// TwinCAT 3 PLC project Untitled1
// ProgramVersion: 3.1.4022.3
// libraries:
//   Tc2_Standard, * (Beckhoff Automation GmbH)
//   Tc2_System, * (Beckhoff Automation GmbH)
//   Tc3_Module, * (Beckhoff Automation GmbH)
// project tree:
//   / PlcTask.TcTTO
//   POUs/ FC1.TcPOU, FC2.TcPOU, FC3.TcPOU, MAIN.TcPOU

CONFIGURATION Untitled1
    RESOURCE PLC ON TwinCAT3
        TASK PlcTask(INTERVAL := T#10ms, PRIORITY := 20);
        PROGRAM MAIN WITH PlcTask : MAIN;
    END_RESOURCE
END_CONFIGURATION

// ---- POUs/MAIN.TcPOU
PROGRAM MAIN
VAR
  test :INT;
  test1 :INT;
  test2 :INT;
  test3 :INT;
  test4 :INT;
END_VAR

END_PROGRAM

// ---- POUs/FC1.TcPOU
PROGRAM FC1
VAR
END_VAR

END_PROGRAM

// ---- POUs/FC2.TcPOU
PROGRAM FC2
VAR
END_VAR

END_PROGRAM

// ---- POUs/FC3.TcPOU
PROGRAM FC3
VAR
END_VAR

END_PROGRAM
